ABB RAPID module: old_Module1.mod

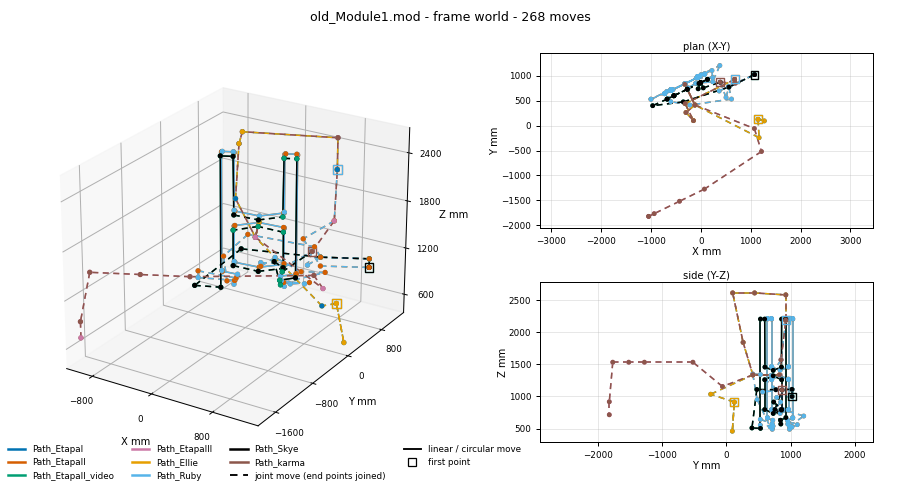
[picture p0: tool path of old_Module1.mod in frame world, 268 of 268 moves have a stored position in this frame; points joined in program order, loops and branches not executed]
MODULE Module1
	CONST robtarget Target_20_2:=[[0,0.000001,500],[0,0,1,-0.000000001],[-2,-1,0,0],[9E9,9E9,9E9,9E9,9E9,9E9]];
	CONST robtarget Target_10:=[[3.472963553,17.439983187,29.999999981],[0,0,1,-0.000000001],[-2,-1,0,0],[9E9,9E9,9E9,9E9,9E9,9E9]];
	CONST robtarget Target_20:=[[0,0.000001,500],[0,0,1,-0.000000001],[-2,-1,0,0],[9E9,9E9,9E9,9E9,9E9,9E9]];
	CONST robtarget Target_20_2_3:=[[355.257254851,-131.298701917,586.23338687],[0,0,1,-0.000000001],[-2,-1,0,0],[9E9,9E9,9E9,9E9,9E9,9E9]];
	CONST robtarget Target_30:=[[-728.668360128,-898.010521018,1225.921750474],[0.579227966,0.405579787,-0.5,-0.5],[0,0,0,0],[9E9,9E9,9E9,9E9,9E9,9E9]];
	CONST robtarget Target_30_3:=[[-1183.134430466,-884.095288461,1304.838955392],[0.579227966,0.405579787,-0.5,-0.5],[1,0,0,0],[9E9,9E9,9E9,9E9,9E9,9E9]];
	CONST robtarget Target_70:=[[-584.684106736,-1037.65235773,1745.210003217],[0.579227966,0.405579787,-0.5,-0.5],[0,0,0,4],[9E9,9E9,9E9,9E9,9E9,9E9]];
	CONST robtarget Target_80_2:=[[-242.789561942,-850.912741716,2444.405198949],[0.579227966,0.405579787,-0.5,-0.5],[1,0,0,4],[9E9,9E9,9E9,9E9,9E9,9E9]];
	CONST robtarget Target_80:=[[-616.524860071,-839.469393295,2509.303652393],[0.69636424,-0.122787804,0,-0.707106781],[0,-1,1,1],[9E9,9E9,9E9,9E9,9E9,9E9]];
	CONST robtarget Target_90:=[[-621.798393161,243.110506611,2288.046539347],[0.69636424,-0.122787804,0,-0.707106781],[0,-1,1,1],[9E9,9E9,9E9,9E9,9E9,9E9]];
	CONST robtarget Target_90_2:=[[-690.279328238,175.6699504,1905.572141463],[0.69636424,-0.122787804,0,-0.707106781],[0,-1,1,1],[9E9,9E9,9E9,9E9,9E9,9E9]];
	CONST robtarget Target_90_2_2:=[[690.970814762,851.051580359,1570.162539077],[0.225435439,0,0,-0.974258109],[0,0,1,1],[9E9,9E9,9E9,9E9,9E9,9E9]];
	CONST robtarget Target_90_2_2_3:=[[367.891360431,693.077349856,1324.929850073],[0,0.848311443,-0.529497588,0],[0,0,-1,0],[9E9,9E9,9E9,9E9,9E9,9E9]];
	CONST robtarget Target_90_2_2_3_2:=[[553.518951213,783.842563864,984.266783155],[0,0.848311443,-0.529497588,0],[0,0,-1,0],[9E9,9E9,9E9,9E9,9E9,9E9]];
	CONST robtarget Target_90_2_2_3_2_2:=[[1075.518835373,1022.097696077,1000],[0,0.848311443,-0.529497588,0],[0,0,-1,0],[9E9,9E9,9E9,9E9,9E9,9E9]];
	CONST robtarget Target_90_2_2_3_2_2_2:=[[1075.518835373,1022.097696077,1000],[0,0.848311443,-0.529497588,0],[0,0,-1,0],[9E9,9E9,9E9,9E9,9E9,9E9]];
	CONST robtarget Target_100:=[[1075.303889935,1021.965880074,1110.91287582],[0,0.848311443,-0.529497588,0],[0,0,-1,0],[9E9,9E9,9E9,9E9,9E9,9E9]];
	CONST robtarget Target_110:=[[561.343174474,770.657579762,1105.422922565],[0,0.848311443,-0.529497588,0],[0,0,-1,0],[9E9,9E9,9E9,9E9,9E9,9E9]];
	CONST robtarget Target_120:=[[614.35326876,531.541624289,1341.660223262],[0.630196274,-0.425266678,-0.564932078,-0.320706495],[0,0,1,0],[9E9,9E9,9E9,9E9,9E9,9E9]];
	CONST robtarget Target_130:=[[-220.756964436,411.144811502,1349.578986688],[0.630196274,-0.425266678,-0.564932078,-0.320706495],[1,1,0,1],[9E9,9E9,9E9,9E9,9E9,9E9]];
	CONST robtarget Target_140:=[[-603.640790819,480.038707024,951.826023694],[0.630196274,-0.425266678,-0.564932078,-0.320706495],[1,0,1,1],[9E9,9E9,9E9,9E9,9E9,9E9]];
	CONST robtarget Target_150:=[[-684.956865831,682.802213826,527.356838346],[0.630196274,-0.425266678,-0.564932078,-0.320706495],[1,0,1,1],[9E9,9E9,9E9,9E9,9E9,9E9]];
	CONST robtarget Target_160:=[[-600.231193595,724.230019574,538.596152517],[0.630196274,-0.425266678,-0.564932078,-0.320706495],[1,0,1,1],[9E9,9E9,9E9,9E9,9E9,9E9]];
	CONST robtarget Target_170:=[[-615.502782618,744.38841834,511.008322261],[0.630196274,-0.425266678,-0.564932078,-0.320706495],[1,0,1,1],[9E9,9E9,9E9,9E9,9E9,9E9]];
	CONST robtarget Target_180:=[[-605.289704553,715.096779867,490.071182954],[0.630196274,-0.425266678,-0.564932078,-0.320706495],[1,0,1,1],[9E9,9E9,9E9,9E9,9E9,9E9]];
	CONST robtarget Target_190:=[[-592.759513668,700.25774586,516.943595123],[0.630196274,-0.425266678,-0.564932078,-0.320706495],[1,0,1,1],[9E9,9E9,9E9,9E9,9E9,9E9]];
	CONST robtarget Target_200:=[[-600.231193595,724.230019574,538.596152517],[0.630196274,-0.425266678,-0.564932078,-0.320706495],[1,0,1,1],[9E9,9E9,9E9,9E9,9E9,9E9]];
	CONST robtarget Target_210:=[[-1000.069986007,528.723234139,554.74513186],[0.630196274,-0.425266678,-0.564932078,-0.320706495],[1,0,1,1],[9E9,9E9,9E9,9E9,9E9,9E9]];
	CONST robtarget Target_210_2:=[[-1000.069986007,528.723234139,644.473462045],[0.74632501,0.144907108,-0.626241041,0.172693565],[1,-1,2,1],[9E9,9E9,9E9,9E9,9E9,9E9]];
	CONST robtarget Target_220:=[[-574.244255672,714.673851005,578.901883612],[0.74632501,0.144907108,-0.626241041,0.172693565],[1,-2,-2,1],[9E9,9E9,9E9,9E9,9E9,9E9]];
	CONST robtarget Target_230:=[[-558.661492442,722.293261641,630.386873665],[0.74632501,0.144907108,-0.626241041,0.172693565],[1,-2,-2,1],[9E9,9E9,9E9,9E9,9E9,9E9]];
	CONST robtarget Target_240:=[[-721.925864829,642.46285692,662.431918782],[0.74632501,0.144907108,-0.626241041,0.172693565],[1,-1,-2,1],[9E9,9E9,9E9,9E9,9E9,9E9]];
	CONST robtarget Target_250:=[[-727.247702444,639.860669777,665.852120215],[0.74632501,0.144907108,-0.626241041,0.172693565],[1,-1,-2,1],[9E9,9E9,9E9,9E9,9E9,9E9]];
	CONST robtarget Target_260:=[[-729.349460263,638.832985813,672.279996312],[0.74632501,0.144907108,-0.626241041,0.172693565],[1,-1,-2,1],[9E9,9E9,9E9,9E9,9E9,9E9]];
	CONST robtarget Target_270:=[[-729.349460263,638.832985813,2203.889],[0.74632501,0.144907108,-0.626241041,0.172693565],[1,-1,-1,1],[9E9,9E9,9E9,9E9,9E9,9E9]];
	CONST robtarget Target_280:=[[-726.718231405,640.119562068,2210.960067812],[0.74632501,0.144907108,-0.626241041,0.172693565],[1,-1,-1,1],[9E9,9E9,9E9,9E9,9E9,9E9]];
	CONST robtarget Target_290:=[[-720.36588301,643.22563191,2213.889],[0.970550763,-0.019647992,0.084912189,0.22457759],[1,0,-2,1],[9E9,9E9,9E9,9E9,9E9,9E9]];
	CONST robtarget Target_300:=[[-603.579378711,700.33003116,2213.889],[0.970550763,-0.019647992,0.084912189,0.22457759],[1,0,-2,1],[9E9,9E9,9E9,9E9,9E9,9E9]];
	CONST robtarget Target_310:=[[-597.227030315,703.436101002,2210.960067812],[0.970550763,-0.019647992,0.084912189,0.22457759],[1,0,-2,1],[9E9,9E9,9E9,9E9,9E9,9E9]];
	CONST robtarget Target_320:=[[-594.595801457,704.722677256,2203.889],[0.970550763,-0.019647992,0.084912189,0.22457759],[1,0,-2,1],[9E9,9E9,9E9,9E9,9E9,9E9]];
	CONST robtarget Target_330:=[[-594.595801457,704.722677256,1467.279996312],[0.970550763,-0.019647992,0.084912189,0.22457759],[1,0,-2,1],[9E9,9E9,9E9,9E9,9E9,9E9]];
	CONST robtarget Target_340:=[[-592.494043638,705.75036122,1460.852120215],[0.970550763,-0.019647992,0.084912189,0.22457759],[1,0,-2,1],[9E9,9E9,9E9,9E9,9E9,9E9]];
	CONST robtarget Target_350:=[[-587.172206023,708.352548362,1457.431918782],[0.970550763,-0.019647992,0.084912189,0.22457759],[1,0,-2,1],[9E9,9E9,9E9,9E9,9E9,9E9]];
	CONST robtarget Target_360:=[[-323.528502026,837.264835131,1406.297094376],[0.970550763,-0.019647992,0.084912189,0.22457759],[1,0,-1,1],[9E9,9E9,9E9,9E9,9E9,9E9]];
	CONST robtarget Target_370:=[[-63.004761668,964.65157192,1457.431918782],[0.970550763,-0.019647992,0.084912189,0.22457759],[1,0,-1,1],[9E9,9E9,9E9,9E9,9E9,9E9]];
	CONST robtarget Target_380:=[[-57.682924053,967.253759063,1460.852120215],[0.970550763,-0.019647992,0.084912189,0.22457759],[1,0,-1,1],[9E9,9E9,9E9,9E9,9E9,9E9]];
	CONST robtarget Target_390:=[[-55.581166233,968.281443027,1467.279996312],[0.970550763,-0.019647992,0.084912189,0.22457759],[1,0,-1,1],[9E9,9E9,9E9,9E9,9E9,9E9]];
	CONST robtarget Target_400:=[[-55.581166233,968.281443027,2203.889],[0.970550763,-0.019647992,0.084912189,0.22457759],[1,0,-1,1],[9E9,9E9,9E9,9E9,9E9,9E9]];
	CONST robtarget Target_410:=[[-52.949937375,969.568019281,2210.960067812],[0.970550763,-0.019647992,0.084912189,0.22457759],[1,0,-1,1],[9E9,9E9,9E9,9E9,9E9,9E9]];
	CONST robtarget Target_420:=[[-46.59758898,972.674089123,2213.889],[0.970550763,-0.019647992,0.084912189,0.22457759],[1,0,-1,1],[9E9,9E9,9E9,9E9,9E9,9E9]];
	CONST robtarget Target_430:=[[70.188915319,1029.778488373,2213.889],[0.970550763,-0.019647992,0.084912189,0.22457759],[0,0,-1,1],[9E9,9E9,9E9,9E9,9E9,9E9]];
	CONST robtarget Target_440:=[[76.541263714,1032.884558215,2210.960067812],[0.970550763,-0.019647992,0.084912189,0.22457759],[0,0,-1,1],[9E9,9E9,9E9,9E9,9E9,9E9]];
	CONST robtarget Target_450:=[[79.172492573,1034.171134469,2203.889],[0.626241041,-0.172693565,0.74632501,0.144907108],[1,1,-2,1],[9E9,9E9,9E9,9E9,9E9,9E9]];
	CONST robtarget Target_460:=[[79.172492573,1034.171134469,672.279996312],[0.626241041,-0.172693565,0.74632501,0.144907108],[1,0,-1,1],[9E9,9E9,9E9,9E9,9E9,9E9]];
	CONST robtarget Target_470:=[[77.070734753,1033.143450506,665.852120215],[0.626241041,-0.172693565,0.74632501,0.144907108],[1,0,-1,1],[9E9,9E9,9E9,9E9,9E9,9E9]];
	CONST robtarget Target_480:=[[71.748897138,1030.541263363,662.431918782],[0.626241041,-0.172693565,0.74632501,0.144907108],[1,0,-1,1],[9E9,9E9,9E9,9E9,9E9,9E9]];
	CONST robtarget Target_490:=[[-91.515475248,950.710858642,630.386873665],[0.626241041,-0.172693565,0.74632501,0.144907108],[1,1,-1,1],[9E9,9E9,9E9,9E9,9E9,9E9]];
	CONST robtarget Target_500:=[[-82.17325952,955.27886605,571.409990938],[0.626241041,-0.172693565,0.74632501,0.144907108],[1,1,-1,1],[9E9,9E9,9E9,9E9,9E9,9E9]];
	CONST robtarget Target_500_2:=[[235.647161917,962.336296138,604.766182313],[0.626241041,-0.172693565,0.74632501,0.144907108],[0,0,-1,1],[9E9,9E9,9E9,9E9,9E9,9E9]];
	CONST robtarget Target_500_2_2:=[[222.398190082,1104.203348059,561.899220237],[0.320706496,-0.564932078,0.425266677,0.630196274],[0,1,-2,0],[9E9,9E9,9E9,9E9,9E9,9E9]];
	CONST robtarget Target_510:=[[4.592265391,1019.966932715,523.466438018],[0.425266678,-0.630196274,0.320706495,0.564932078],[0,1,-2,0],[9E9,9E9,9E9,9E9,9E9,9E9]];
	CONST robtarget Target_520:=[[-67.51635848,984.708409724,538.596152517],[0.425266678,-0.630196274,0.320706495,0.564932078],[0,1,-2,0],[9E9,9E9,9E9,9E9,9E9,9E9]];
	CONST robtarget Target_530:=[[-74.04786326,1009.140395264,511.008322261],[0.425266678,-0.630196274,0.320706495,0.564932078],[0,1,-2,0],[9E9,9E9,9E9,9E9,9E9,9E9]];
	CONST robtarget Target_540:=[[-57.20170243,983.09209564,490.071182954],[0.425266678,-0.630196274,0.320706495,0.564932078],[0,1,-2,0],[9E9,9E9,9E9,9E9,9E9,9E9]];
	CONST robtarget Target_550:=[[-53.184944606,964.090299134,516.943595123],[0.425266678,-0.630196274,0.320706495,0.564932078],[0,1,-2,0],[9E9,9E9,9E9,9E9,9E9,9E9]];
	CONST robtarget Target_560:=[[-67.51635848,984.708409724,538.596152517],[0.425266678,-0.630196274,0.320706495,0.564932078],[0,1,-2,0],[9E9,9E9,9E9,9E9,9E9,9E9]];
	CONST robtarget Target_570:=[[380.563228786,1203.803208398,695.774665043],[0.425266678,-0.630196274,0.320706495,0.564932078],[0,1,-2,0],[9E9,9E9,9E9,9E9,9E9,9E9]];
	CONST robtarget Target_580_3:=[[236.855316057,878.977367128,797.279996312],[0.626241041,-0.172693565,0.74632501,0.144907108],[0,0,-1,1],[9E9,9E9,9E9,9E9,9E9,9E9]];
	CONST robtarget Target_740:=[[-106.574951523,844.917671275,913.754533399],[0.626241041,-0.172693565,0.74632501,0.144907108],[1,1,-1,1],[9E9,9E9,9E9,9E9,9E9,9E9]];
	CONST robtarget Target_580_3_2:=[[-251.957733199,755.881530829,797.279996312],[0.626241041,-0.172693565,0.74632501,0.144907108],[1,1,-1,1],[9E9,9E9,9E9,9E9,9E9,9E9]];
	CONST robtarget Target_580:=[[-306.602704629,845.540941159,797.279996312],[0.626241041,-0.172693565,0.74632501,0.144907108],[1,1,-1,1],[9E9,9E9,9E9,9E9,9E9,9E9]];
	CONST robtarget Target_590:=[[-55.581166233,968.281443027,797.279996312],[0.626241041,-0.172693565,0.74632501,0.144907108],[1,1,-1,1],[9E9,9E9,9E9,9E9,9E9,9E9]];
	CONST robtarget Target_600:=[[-55.581166233,968.281443027,1260.498003688],[0.626241041,-0.172693565,0.74632501,0.144907108],[1,1,-1,1],[9E9,9E9,9E9,9E9,9E9,9E9]];
	CONST robtarget Target_610:=[[-57.682924053,967.253759063,1266.925879785],[0.626241041,-0.172693565,0.74632501,0.144907108],[1,1,-1,1],[9E9,9E9,9E9,9E9,9E9,9E9]];
	CONST robtarget Target_620:=[[-63.004761668,964.65157192,1270.346081218],[0.626241041,-0.172693565,0.74632501,0.144907108],[1,1,-1,1],[9E9,9E9,9E9,9E9,9E9,9E9]];
	CONST robtarget Target_630:=[[-326.648465665,835.739285151,1321.480905624],[0.626241041,-0.172693565,0.74632501,0.144907108],[1,1,-1,1],[9E9,9E9,9E9,9E9,9E9,9E9]];
	CONST robtarget Target_640:=[[-587.172206023,708.352548362,1270.346081218],[0.626241041,-0.172693565,0.74632501,0.144907108],[1,1,-1,1],[9E9,9E9,9E9,9E9,9E9,9E9]];
	CONST robtarget Target_650:=[[-592.494043638,705.75036122,1266.925879785],[0.626241041,-0.172693565,0.74632501,0.144907108],[1,1,-1,1],[9E9,9E9,9E9,9E9,9E9,9E9]];
	CONST robtarget Target_660:=[[-594.595801457,704.722677256,1260.498003688],[0.626241041,-0.172693565,0.74632501,0.144907108],[1,1,-1,1],[9E9,9E9,9E9,9E9,9E9,9E9]];
	CONST robtarget Target_670:=[[-594.595801457,704.722677256,797.279996312],[0.626241041,-0.172693565,0.74632501,0.144907108],[1,1,-1,1],[9E9,9E9,9E9,9E9,9E9,9E9]];
	CONST robtarget Target_680:=[[-592.494043638,705.75036122,790.852120215],[0.626241041,-0.172693565,0.74632501,0.144907108],[1,1,-1,1],[9E9,9E9,9E9,9E9,9E9,9E9]];
	CONST robtarget Target_690:=[[-587.172206023,708.352548362,787.431918782],[0.626241041,-0.172693565,0.74632501,0.144907108],[1,1,-1,1],[9E9,9E9,9E9,9E9,9E9,9E9]];
	CONST robtarget Target_700:=[[-323.528502026,837.264835131,736.297094376],[0.626241041,-0.172693565,0.74632501,0.144907108],[1,1,-1,1],[9E9,9E9,9E9,9E9,9E9,9E9]];
	CONST robtarget Target_710:=[[-63.004761668,964.65157192,787.431918782],[0.626241041,-0.172693565,0.74632501,0.144907108],[1,1,-1,1],[9E9,9E9,9E9,9E9,9E9,9E9]];
	CONST robtarget Target_720:=[[-57.682924053,967.253759063,790.852120215],[0.626241041,-0.172693565,0.74632501,0.144907108],[1,1,-1,1],[9E9,9E9,9E9,9E9,9E9,9E9]];
	CONST robtarget Target_730:=[[-55.581166233,968.281443027,797.279996312],[0.626241041,-0.172693565,0.74632501,0.144907108],[1,1,-1,1],[9E9,9E9,9E9,9E9,9E9,9E9]];
	CONST robtarget Target_730_2:=[[-4.129380996,863.055327059,797.279996312],[0.626241041,-0.172693565,0.74632501,0.144907108],[1,1,-1,1],[9E9,9E9,9E9,9E9,9E9,9E9]];
	CONST robtarget Target_130_2:=[[389.997020927,869.040623857,1101.572770211],[0.630196274,-0.425266678,-0.564932078,-0.320706495],[0,1,0,0],[9E9,9E9,9E9,9E9,9E9,9E9]];
	CONST robtarget Target_120_2:=[[504.928038476,563.849286682,1069.091100494],[0,0.848311443,-0.529497588,0],[0,0,-1,0],[9E9,9E9,9E9,9E9,9E9,9E9]];
	CONST robtarget Target_110_2:=[[561.343174474,770.657579762,1105.422922565],[0,0.848311443,-0.529497588,0],[0,0,-1,0],[9E9,9E9,9E9,9E9,9E9,9E9]];
	CONST robtarget Target_90_2_2_3_2_2_2_2:=[[1075.518835373,1022.097696077,1000],[0,0.848311443,-0.529497588,0],[0,0,-1,0],[9E9,9E9,9E9,9E9,9E9,9E9]];
	CONST robtarget Target_100_2:=[[1075.303889935,1021.965880074,1110.91287582],[0,0.848311443,-0.529497588,0],[0,0,-1,0],[9E9,9E9,9E9,9E9,9E9,9E9]];
	CONST robtarget Target_110_3:=[[561.343174474,770.657579762,1105.422922565],[0,0.848311443,-0.529497588,0],[0,0,-1,0],[9E9,9E9,9E9,9E9,9E9,9E9]];
	CONST robtarget Target_120_3:=[[-352.181570531,474.725664361,1108.429867517],[0.630196274,-0.425266678,-0.564932078,-0.320706495],[1,-2,-1,0],[9E9,9E9,9E9,9E9,9E9,9E9]];
	CONST robtarget Target_130_3:=[[-965.595492909,398.655755176,510.210088752],[0.630196274,-0.425266678,-0.564932078,-0.320706495],[1,-2,-1,0],[9E9,9E9,9E9,9E9,9E9,9E9]];
	CONST robtarget Target_260_2:=[[-676.765426106,531.291262028,504.173173014],[0.630196274,-0.425266678,-0.564932078,-0.320706495],[1,-2,-1,0],[9E9,9E9,9E9,9E9,9E9,9E9]];
	CONST robtarget Target_270_2:=[[-676.765426106,531.291262028,2203.889],[0.630196274,-0.425266678,-0.564932078,-0.320706495],[1,-1,-2,0],[9E9,9E9,9E9,9E9,9E9,9E9]];
	CONST robtarget Target_320_2:=[[-542.0117673,597.180953471,2203.889],[0.630196274,-0.425266678,-0.564932078,-0.320706495],[1,-1,-2,0],[9E9,9E9,9E9,9E9,9E9,9E9]];
	CONST robtarget Target_350_2:=[[-534.588171866,600.810824577,1457.431918782],[0.630196274,-0.425266678,-0.564932078,-0.320706495],[1,-1,-1,0],[9E9,9E9,9E9,9E9,9E9,9E9]];
	CONST robtarget Target_360_2:=[[-270.944467869,729.723111346,1406.297094376],[0.630196274,-0.425266678,-0.564932078,-0.320706495],[1,-1,-1,1],[9E9,9E9,9E9,9E9,9E9,9E9]];
	CONST robtarget Target_370_2:=[[-10.420727511,857.109848135,1457.431918782],[0.630196274,-0.425266678,-0.564932078,-0.320706495],[0,-1,-1,1],[9E9,9E9,9E9,9E9,9E9,9E9]];
	CONST robtarget Target_400_2:=[[-2.997132076,860.739719242,2203.889],[0.630196274,-0.425266678,-0.564932078,-0.320706495],[0,-2,-1,1],[9E9,9E9,9E9,9E9,9E9,9E9]];
	CONST robtarget Target_450_2:=[[131.75652673,926.629410684,2203.889],[0.630196274,-0.425266678,-0.564932078,-0.320706495],[0,-2,-1,1],[9E9,9E9,9E9,9E9,9E9,9E9]];
	CONST robtarget Target_460_2:=[[131.75652673,926.629410684,672.279996312],[0.630196274,-0.425266678,-0.564932078,-0.320706495],[0,-1,-2,1],[9E9,9E9,9E9,9E9,9E9,9E9]];
	CONST robtarget Target_490_2:=[[-38.931441091,843.169134857,630.386873665],[0.630196274,-0.425266678,-0.564932078,-0.320706495],[0,-1,-2,1],[9E9,9E9,9E9,9E9,9E9,9E9]];
	CONST robtarget Target_500_3:=[[-29.589225363,847.737142265,571.409990938],[0.630196274,-0.425266678,-0.564932078,-0.320706495],[0,-1,-2,1],[9E9,9E9,9E9,9E9,9E9,9E9]];
	CONST robtarget Target_740_2:=[[-53.990917366,737.37594749,913.754533399],[0.630196274,-0.425266678,-0.564932078,-0.320706495],[0,-1,-2,1],[9E9,9E9,9E9,9E9,9E9,9E9]];
	CONST robtarget Target_590_2:=[[-2.997132076,860.739719242,797.279996312],[0.630196274,-0.425266678,-0.564932078,-0.320706495],[0,-1,-2,1],[9E9,9E9,9E9,9E9,9E9,9E9]];
	CONST robtarget Target_600_2:=[[-2.997132076,860.739719242,1260.498003688],[0.630196274,-0.425266678,-0.564932078,-0.320706495],[0,-1,-2,1],[9E9,9E9,9E9,9E9,9E9,9E9]];
	CONST robtarget Target_630_2:=[[-274.064431508,728.197561366,1321.480905624],[0.630196274,-0.425266678,-0.564932078,-0.320706495],[1,-1,-2,1],[9E9,9E9,9E9,9E9,9E9,9E9]];
	CONST robtarget Target_660_2:=[[-542.0117673,597.180953471,1260.498003688],[0.630196274,-0.425266678,-0.564932078,-0.320706495],[1,-2,-1,0],[9E9,9E9,9E9,9E9,9E9,9E9]];
	CONST robtarget Target_670_2:=[[-542.0117673,597.180953471,797.279996312],[0.630196274,-0.425266678,-0.564932078,-0.320706495],[1,-2,-1,0],[9E9,9E9,9E9,9E9,9E9,9E9]];
	CONST robtarget Target_700_2:=[[-270.944467869,729.723111346,736.297094376],[0.630196274,-0.425266678,-0.564932078,-0.320706495],[1,-1,-2,1],[9E9,9E9,9E9,9E9,9E9,9E9]];
	CONST robtarget Target_710_2:=[[-10.420727511,857.109848135,787.431918782],[0.630196274,-0.425266678,-0.564932078,-0.320706495],[0,-1,-2,1],[9E9,9E9,9E9,9E9,9E9,9E9]];
	CONST robtarget Target_730_3:=[[-2.997132076,860.739719242,797.279996312],[0.630196274,-0.425266678,-0.564932078,-0.320706495],[0,-1,-2,1],[9E9,9E9,9E9,9E9,9E9,9E9]];
	CONST robtarget Target_730_2_2:=[[48.454653161,755.513603274,797.279996312],[0.630196274,-0.425266678,-0.564932078,-0.320706495],[0,-1,-2,1],[9E9,9E9,9E9,9E9,9E9,9E9]];
	CONST robtarget Target_130_2_2:=[[389.997020927,869.040623857,1101.572770211],[0.630196274,-0.425266678,-0.564932078,-0.320706495],[0,-1,-2,1],[9E9,9E9,9E9,9E9,9E9,9E9]];
	CONST robtarget Target_130_2_2_2:=[[389.997020927,869.040623857,1101.572770211],[0.630196274,-0.425266678,-0.564932078,-0.320706495],[0,-1,-2,1],[9E9,9E9,9E9,9E9,9E9,9E9]];
	CONST robtarget Target_90_2_2_2:=[[690.970814762,851.051580359,1570.162539077],[0.225435439,0,0,-0.974258109],[0,0,1,1],[9E9,9E9,9E9,9E9,9E9,9E9]];
	CONST robtarget Target_90_2_3:=[[677.216886302,925.105208889,2185.609751442],[0.225435439,0,0,-0.974258109],[0,0,1,1],[9E9,9E9,9E9,9E9,9E9,9E9]];
	CONST robtarget Target_90_2_4:=[[677.216886302,925.105208889,2185.609751442],[0.225435439,0,0,-0.974258109],[0,0,1,1],[9E9,9E9,9E9,9E9,9E9,9E9]];
	CONST robtarget Target_90_3:=[[677.216886303,925.105208888,2579.975738982],[0.225435439,0,0,-0.974258109],[0,0,1,1],[9E9,9E9,9E9,9E9,9E9,9E9]];
	CONST robtarget Target_80_3:=[[-315.067708607,439.913739054,2610.344805668],[0.225435439,0,0,-0.974258109],[1,0,0,1],[9E9,9E9,9E9,9E9,9E9,9E9]];
	CONST robtarget Target_80_2_2:=[[-148.366452112,98.986292765,2610.344805667],[0.159406928,0.159406928,-0.688904515,-0.688904516],[1,0,0,4],[9E9,9E9,9E9,9E9,9E9,9E9]];
	CONST robtarget Target_70_2:=[[-297.408117168,261.539979913,1840.929204997],[0.159406928,0.159406928,-0.688904515,-0.688904516],[0,0,0,4],[9E9,9E9,9E9,9E9,9E9,9E9]];
	CONST robtarget Target_30_2:=[[-117.985307131,412.947477324,1336.176966578],[0.159406928,0.159406928,-0.688904515,-0.688904516],[0,0,0,0],[9E9,9E9,9E9,9E9,9E9,9E9]];
	CONST robtarget Target_30_3_2:=[[-320.695795916,827.518853271,1336.176966578],[0.159406928,0.159406928,-0.688904515,-0.688904516],[1,0,0,0],[9E9,9E9,9E9,9E9,9E9,9E9]];
	CONST robtarget Target_30_2_2:=[[-117.985307131,412.947477324,1336.176966578],[0.159406928,0.159406928,-0.688904515,-0.688904516],[0,0,0,0],[9E9,9E9,9E9,9E9,9E9,9E9]];
	CONST robtarget Target_30_2_3:=[[1072.781898944,-59.825918958,1155.239486671],[0.374411334,0.374411335,0.599846774,0.599846775],[-1,1,-1,0],[9E9,9E9,9E9,9E9,9E9,9E9]];
	CONST robtarget Target_30_2_3_2:=[[1215.425844801,-519.48484737,1533.087792477],[0.374411334,0.374411335,0.599846774,0.599846775],[-1,1,-1,0],[9E9,9E9,9E9,9E9,9E9,9E9]];
	CONST robtarget Target_30_2_3_2_2:=[[71.368530681,-1273.53877769,1533.087792477],[0.688904515,0.688904516,0.159406928,0.159406928],[-2,1,-1,0],[9E9,9E9,9E9,9E9,9E9,9E9]];
	CONST robtarget Target_30_2_3_2_2_2:=[[-427.431513587,-1517.434055188,1533.087792477],[0.000000001,0.974258109,0.225435439,0],[-2,-1,0,0],[9E9,9E9,9E9,9E9,9E9,9E9]];
	CONST robtarget Target_30_2_3_2_2_2_2:=[[-935.838539063,-1766.02680089,1533.087792477],[-0.000000001,0.974258109,0.225435439,0],[-2,0,0,0],[9E9,9E9,9E9,9E9,9E9,9E9]];
	CONST robtarget Target_30_2_3_2_2_2_2_2:=[[-1046.370183316,-1820.072798594,917.887564527],[-0.000000001,0.974258109,0.225435439,0],[-2,0,0,0],[9E9,9E9,9E9,9E9,9E9,9E9]];
	CONST robtarget Target_30_2_3_2_2_2_2_2_2:=[[-1046.370183316,-1820.072798594,715.608584776],[-0.000000001,0.974258109,0.225435439,0],[-2,0,0,0],[9E9,9E9,9E9,9E9,9E9,9E9]];
	PROC Path_EtapaI()
	    MoveJ Target_20_2,v500,z100,Tooldata_TCP_VAC\WObj:=Workobject_EtapaI;
	    MoveJ Target_10,v400,z100,Tooldata_TCP_VAC\WObj:=Workobject_EtapaI;
	    MoveJ Target_20,v500,z100,Tooldata_TCP_VAC\WObj:=Workobject_EtapaI;
	    MoveJ Target_20_2_3,v500,z100,Tooldata_TCP_VAC\WObj:=Workobject_EtapaI;
	    MoveJ Target_30,v500,z100,Tooldata_TCP_VAC\WObj:=Workobject_EtapaI;
	    MoveJ Target_30_3,v500,z100,Tooldata_TCP_VAC\WObj:=Workobject_EtapaI;
	    MoveJ Target_30,v500,z100,Tooldata_TCP_VAC\WObj:=Workobject_EtapaI;
	    MoveJ Target_70,v500,z100,Tooldata_TCP_VAC\WObj:=Workobject_EtapaI;
	    MoveJ Target_80_2,v500,z100,Tooldata_TCP_VAC\WObj:=Workobject_EtapaI;
	    MoveJ Target_80,v500,z100,Tooldata_TCP_VAC\WObj:=Workobject_EtapaI;
	    MoveJ Target_90,v500,z100,Tooldata_TCP_VAC\WObj:=Workobject_EtapaI;
	    MoveJ Target_90_2,v500,z100,Tooldata_TCP_VAC\WObj:=Workobject_EtapaI;
	ENDPROC
	PROC Path_EtapaII()
	    MoveJ Target_90_2,v500,z100,Tooldata_TCP_VAC\WObj:=Workobject_EtapaI;
	    MoveJ Target_90_2_2,v500,z100,Flansa_Cuplare\WObj:=Workobject_EtapaII;
	    MoveJ Target_90_2_2_3,v500,z100,Flansa_Cuplare\WObj:=Workobject_EtapaII;
	    MoveJ Target_90_2_2_3_2,v500,z100,Flansa_Cuplare\WObj:=Workobject_EtapaII;
	    MoveJ Target_90_2_2_3_2_2,v500,z100,Flansa_Cuplare\WObj:=Workobject_EtapaII;
	    MoveJ Target_90_2_2_3_2_2_2,v500,z100,Flansa_Cuplare\WObj:=Workobject_EtapaII;
	    MoveJ Target_100,v500,z100,Flansa_Cuplare\WObj:=Workobject_EtapaII;
	    MoveJ Target_110,v500,z100,Flansa_Cuplare\WObj:=Workobject_EtapaII;
	    MoveJ Target_120,v500,z100,Flansa_Cuplare\WObj:=Workobject_EtapaII;
	    MoveJ Target_130,v500,z100,Flansa_Cuplare\WObj:=Workobject_EtapaII;
	    MoveJ Target_140,v500,z100,Flansa_Cuplare\WObj:=Workobject_EtapaII;
	    MoveJ Target_150,v1000,z100,Tooldata_TCP_ATI\WObj:=Workobject_EtapaII;
	    MoveJ Target_160,v1000,z100,Tooldata_TCP_ATI\WObj:=Workobject_EtapaII;
	    MoveC Target_170,Target_180,v1000,z100,Tooldata_TCP_ATI\WObj:=Workobject_EtapaII;
	    MoveC Target_190,Target_200,v1000,z100,Tooldata_TCP_ATI\WObj:=Workobject_EtapaII;
	    MoveJ Target_210,v1000,z100,Tooldata_TCP_ATI\WObj:=Workobject_EtapaII;
	    MoveJ Target_210_2,v1000,z100,Tooldata_TCP_ATI\WObj:=Workobject_EtapaII;
	    MoveJ Target_220,v1000,z100,Tooldata_TCP_ATI\WObj:=Workobject_EtapaII;
	    MoveL Target_230,v1000,z100,Tooldata_TCP_ATI\WObj:=Workobject_EtapaII;
	    MoveL Target_240,v1000,z100,Tooldata_TCP_ATI\WObj:=Workobject_EtapaII;
	    MoveL Target_250,v1000,z100,Tooldata_TCP_ATI\WObj:=Workobject_EtapaII;
	    MoveL Target_260,v1000,z100,Tooldata_TCP_ATI\WObj:=Workobject_EtapaII;
	    MoveL Target_270,v1000,z100,Tooldata_TCP_ATI\WObj:=Workobject_EtapaII;
	    MoveL Target_280,v1000,z100,Tooldata_TCP_ATI\WObj:=Workobject_EtapaII;
	    MoveL Target_290,v1000,z100,Tooldata_TCP_ATI\WObj:=Workobject_EtapaII;
	    MoveL Target_300,v1000,z100,Tooldata_TCP_ATI\WObj:=Workobject_EtapaII;
	    MoveL Target_310,v1000,z100,Tooldata_TCP_ATI\WObj:=Workobject_EtapaII;
	    MoveL Target_320,v1000,z100,Tooldata_TCP_ATI\WObj:=Workobject_EtapaII;
	    MoveL Target_330,v1000,z100,Tooldata_TCP_ATI\WObj:=Workobject_EtapaII;
	    MoveL Target_340,v1000,z100,Tooldata_TCP_ATI\WObj:=Workobject_EtapaII;
	    MoveL Target_350,v1000,z100,Tooldata_TCP_ATI\WObj:=Workobject_EtapaII;
	    MoveL Target_360,v1000,z100,Tooldata_TCP_ATI\WObj:=Workobject_EtapaII;
	    MoveL Target_370,v1000,z100,Tooldata_TCP_ATI\WObj:=Workobject_EtapaII;
	    MoveL Target_380,v1000,z100,Tooldata_TCP_ATI\WObj:=Workobject_EtapaII;
	    MoveL Target_390,v1000,z100,Tooldata_TCP_ATI\WObj:=Workobject_EtapaII;
	    MoveL Target_400,v1000,z100,Tooldata_TCP_ATI\WObj:=Workobject_EtapaII;
	    MoveL Target_410,v1000,z100,Tooldata_TCP_ATI\WObj:=Workobject_EtapaII;
	    MoveL Target_420,v1000,z100,Tooldata_TCP_ATI\WObj:=Workobject_EtapaII;
	    MoveL Target_430,v1000,z100,Tooldata_TCP_ATI\WObj:=Workobject_EtapaII;
	    MoveJ Target_440,v1000,z100,Tooldata_TCP_ATI\WObj:=Workobject_EtapaII;
	    MoveJ Target_450,v1000,z100,Tooldata_TCP_ATI\WObj:=Workobject_EtapaII;
	    MoveL Target_460,v1000,z100,Tooldata_TCP_ATI\WObj:=Workobject_EtapaII;
	    MoveL Target_470,v1000,z100,Tooldata_TCP_ATI\WObj:=Workobject_EtapaII;
	    MoveL Target_480,v1000,z100,Tooldata_TCP_ATI\WObj:=Workobject_EtapaII;
	    MoveL Target_490,v1000,z100,Tooldata_TCP_ATI\WObj:=Workobject_EtapaII;
	    MoveL Target_500,v1000,z100,Tooldata_TCP_ATI\WObj:=Workobject_EtapaII;
	    MoveJ Target_500_2,v1000,z100,Tooldata_TCP_ATI\WObj:=Workobject_EtapaII;
	    MoveJ Target_500_2_2,v1000,z100,Tooldata_TCP_ATI\WObj:=Workobject_EtapaII;
	    MoveJ Target_510,v1000,z100,Tooldata_TCP_ATI\WObj:=Workobject_EtapaII;
	    MoveJ Target_520,v1000,z100,Tooldata_TCP_ATI\WObj:=Workobject_EtapaII;
	    MoveC Target_530,Target_540,v1000,z100,Tooldata_TCP_ATI\WObj:=Workobject_EtapaII;
	    MoveC Target_550,Target_560,v1000,z100,Tooldata_TCP_ATI\WObj:=Workobject_EtapaII;
	    MoveJ Target_570,v1000,z100,Tooldata_TCP_ATI\WObj:=Workobject_EtapaII;
	    MoveJ Target_580_3,v1000,z100,Tooldata_TCP_ATI\WObj:=Workobject_EtapaII;
	    MoveJ Target_740,v1000,z100,Tooldata_TCP_ATI\WObj:=Workobject_EtapaII;
	    MoveJ Target_580_3_2,v1000,z100,Tooldata_TCP_ATI\WObj:=Workobject_EtapaII;
	    MoveJ Target_580,v1000,z100,Tooldata_TCP_ATI\WObj:=Workobject_EtapaII;
	    MoveJ Target_590,v1000,z100,Tooldata_TCP_ATI\WObj:=Workobject_EtapaII;
	    MoveL Target_600,v1000,z100,Tooldata_TCP_ATI\WObj:=Workobject_EtapaII;
	    MoveL Target_610,v1000,z100,Tooldata_TCP_ATI\WObj:=Workobject_EtapaII;
	    MoveL Target_620,v1000,z100,Tooldata_TCP_ATI\WObj:=Workobject_EtapaII;
	    MoveL Target_630,v1000,z100,Tooldata_TCP_ATI\WObj:=Workobject_EtapaII;
	    MoveL Target_640,v1000,z100,Tooldata_TCP_ATI\WObj:=Workobject_EtapaII;
	    MoveL Target_650,v1000,z100,Tooldata_TCP_ATI\WObj:=Workobject_EtapaII;
	    MoveL Target_660,v1000,z100,Tooldata_TCP_ATI\WObj:=Workobject_EtapaII;
	    MoveL Target_670,v1000,z100,Tooldata_TCP_ATI\WObj:=Workobject_EtapaII;
	    MoveL Target_680,v1000,z100,Tooldata_TCP_ATI\WObj:=Workobject_EtapaII;
	    MoveL Target_690,v1000,z100,Tooldata_TCP_ATI\WObj:=Workobject_EtapaII;
	    MoveL Target_700,v1000,z100,Tooldata_TCP_ATI\WObj:=Workobject_EtapaII;
	    MoveL Target_710,v1000,z100,Tooldata_TCP_ATI\WObj:=Workobject_EtapaII;
	    MoveL Target_720,v1000,z100,Tooldata_TCP_ATI\WObj:=Workobject_EtapaII;
	    MoveL Target_730,v1000,z100,Tooldata_TCP_ATI\WObj:=Workobject_EtapaII;
	    MoveJ Target_730_2,v1000,z100,Tooldata_TCP_ATI\WObj:=Workobject_EtapaII;
	    MoveJ Target_130_2,v500,z100,Flansa_Cuplare\WObj:=Workobject_EtapaII;
	    MoveJ Target_120_2,v500,z100,Flansa_Cuplare\WObj:=Workobject_EtapaII;
	    MoveJ Target_110_2,v500,z100,Flansa_Cuplare\WObj:=Workobject_EtapaII;
	    MoveJ Target_100,v500,z100,Flansa_Cuplare\WObj:=Workobject_EtapaII;
	ENDPROC
	PROC Path_EtapaII_video()
	    MoveJ Target_90_2_2_3_2_2_2_2,v500,z100,Flansa_Cuplare\WObj:=Workobject_EtapaII_video;
	    MoveJ Target_100_2,v500,z100,Flansa_Cuplare\WObj:=Workobject_EtapaII_video;
	    MoveJ Target_110_3,v500,z100,Flansa_Cuplare\WObj:=Workobject_EtapaII_video;
	    MoveJ Target_120_3,v500,z100,Flansa_Cuplare\WObj:=Workobject_EtapaII_video;
	    MoveJ Target_130_3,v500,z50,Flansa_Cuplare\WObj:=Workobject_EtapaII_video;
	    MoveJ Target_260_2,v100,z50,Flansa_Cuplare\WObj:=Workobject_EtapaII_video;
	    MoveL Target_270_2,v200,z50,Flansa_Cuplare\WObj:=Workobject_EtapaII_video;
	    MoveL Target_320_2,v1000,z100,Flansa_Cuplare\WObj:=Workobject_EtapaII_video;
	    MoveL Target_350_2,v300,z30,Flansa_Cuplare\WObj:=Workobject_EtapaII_video;
	    MoveJ Target_360_2,v300,z30,Flansa_Cuplare\WObj:=Workobject_EtapaII_video;
	    MoveJ Target_370_2,v300,z30,Flansa_Cuplare\WObj:=Workobject_EtapaII_video;
	    MoveL Target_400_2,v300,z30,Flansa_Cuplare\WObj:=Workobject_EtapaII_video;
	    MoveJ Target_450_2,v300,z30,Flansa_Cuplare\WObj:=Workobject_EtapaII_video;
	    MoveL Target_460_2,v300,z30,Flansa_Cuplare\WObj:=Workobject_EtapaII_video;
	    MoveL Target_490_2,v300,z30,Flansa_Cuplare\WObj:=Workobject_EtapaII_video;
	    MoveL Target_500_3,v300,z30,Flansa_Cuplare\WObj:=Workobject_EtapaII_video;
	    MoveJ Target_740_2,v400,z20,Flansa_Cuplare\WObj:=Workobject_EtapaII_video;
	    MoveJ Target_590_2,v300,z30,Flansa_Cuplare\WObj:=Workobject_EtapaII_video;
	    MoveL Target_600_2,v300,z30,Flansa_Cuplare\WObj:=Workobject_EtapaII_video;
	    MoveJ Target_630_2,v300,z30,Flansa_Cuplare\WObj:=Workobject_EtapaII_video;
	    MoveJ Target_660_2,v300,z30,Flansa_Cuplare\WObj:=Workobject_EtapaII_video;
	    MoveL Target_670_2,v300,z30,Flansa_Cuplare\WObj:=Workobject_EtapaII_video;
	    MoveJ Target_700_2,v300,z30,Flansa_Cuplare\WObj:=Workobject_EtapaII_video;
	    MoveJ Target_710_2,v300,z30,Flansa_Cuplare\WObj:=Workobject_EtapaII_video;
	    MoveL Target_730_3,v300,z30,Flansa_Cuplare\WObj:=Workobject_EtapaII_video;
	    MoveJ Target_730_2_2,v300,z30,Flansa_Cuplare\WObj:=Workobject_EtapaII_video;
	    MoveJ Target_130_2_2,v300,z30,Flansa_Cuplare\WObj:=Workobject_EtapaII_video;
	ENDPROC
	PROC Path_EtapaIII()
	    MoveJ Target_130_2_2_2,v400,z30,Flansa_Cuplare\WObj:=Workobject_EtapaIII;
	    MoveJ Target_90_2_2_2,v400,z30,Flansa_Cuplare\WObj:=Workobject_EtapaIII;
	    MoveJ Target_90_2_3,v400,z30,Tooldata_TCP_VAC\WObj:=Workobject_EtapaIII;
	    MoveJ Target_90_2_4,v400,z30,Tooldata_TCP_VAC\WObj:=Workobject_EtapaIII;
	    MoveJ Target_90_3,v400,z30,Tooldata_TCP_VAC\WObj:=Workobject_EtapaIII;
	    MoveJ Target_80_3,v400,z30,Tooldata_TCP_VAC\WObj:=Workobject_EtapaIII;
	    MoveJ Target_80_2_2,v400,z30,Tooldata_TCP_VAC\WObj:=Workobject_EtapaIII;
	    MoveJ Target_70_2,v400,z30,Tooldata_TCP_VAC\WObj:=Workobject_EtapaIII;
	    MoveJ Target_30_2,v150,z10,Tooldata_TCP_VAC\WObj:=Workobject_EtapaIII;
	    MoveL Target_30_3_2,v150,z10,Tooldata_TCP_VAC\WObj:=Workobject_EtapaIII;
	    MoveL Target_30_2_2,v150,z10,Tooldata_TCP_VAC\WObj:=Workobject_EtapaIII;
	    MoveJ Target_30_2_3,v300,z30,Tooldata_TCP_VAC\WObj:=Workobject_EtapaIII;
	    MoveJ Target_30_2_3_2,v300,z30,Tooldata_TCP_VAC\WObj:=Workobject_EtapaIII;
	    MoveJ Target_30_2_3_2_2,v300,z30,Tooldata_TCP_VAC\WObj:=Workobject_EtapaIII;
	    MoveJ Target_30_2_3_2_2_2,v300,z30,Tooldata_TCP_VAC\WObj:=Workobject_EtapaIII;
	    MoveJ Target_30_2_3_2_2_2_2,v300,z30,Tooldata_TCP_VAC\WObj:=Workobject_EtapaIII;
	    MoveJ Target_30_2_3_2_2_2_2_2,v300,z30,Tooldata_TCP_VAC\WObj:=Workobject_EtapaIII;
	    MoveJ Target_30_2_3_2_2_2_2_2_2,v300,z30,Tooldata_TCP_VAC\WObj:=Workobject_EtapaIII;
	ENDPROC
	PROC Path_10()

	ENDPROC
	PROC Path_Ellie()
	    MoveJ Target_20_2,v500,z100,Tooldata_TCP_VAC\WObj:=Workobject_ellie;
	    MoveJ Target_10,v400,z100,Tooldata_TCP_VAC\WObj:=Workobject_ellie;
	    MoveJ Target_20,v500,z100,Tooldata_TCP_VAC\WObj:=Workobject_ellie;
	    MoveJ Target_20_2_3,v500,z100,Tooldata_TCP_VAC\WObj:=Workobject_ellie;
	    MoveJ Target_30,v500,z100,Tooldata_TCP_VAC\WObj:=Workobject_ellie;
	    MoveJ Target_30_3,v500,z100,Tooldata_TCP_VAC\WObj:=Workobject_ellie;
	    MoveJ Target_30,v500,z100,Tooldata_TCP_VAC\WObj:=Workobject_ellie;
	    MoveJ Target_70,v500,z100,Tooldata_TCP_VAC\WObj:=Workobject_ellie;
	    MoveJ Target_80_2,v500,z100,Tooldata_TCP_VAC\WObj:=Workobject_ellie;
	    MoveJ Target_80,v500,z100,Tooldata_TCP_VAC\WObj:=Workobject_ellie;
	    MoveJ Target_90,v500,z100,Tooldata_TCP_VAC\WObj:=Workobject_ellie;
	    MoveJ Target_90_2,v500,z100,Tooldata_TCP_VAC\WObj:=Workobject_ellie;
	ENDPROC
	PROC Path_Ruby()
	    MoveJ Target_90_2,v500,z100,Tooldata_TCP_VAC\WObj:=Workobject_ellie;
	    MoveJ Target_90_2_2,v500,z100,Flansa_Cuplare\WObj:=Workobject_ruby;
	    MoveJ Target_90_2_2_3,v500,z100,Flansa_Cuplare\WObj:=Workobject_ruby;
	    MoveJ Target_90_2_2_3_2,v500,z100,Flansa_Cuplare\WObj:=Workobject_ruby;
	    MoveJ Target_90_2_2_3_2_2,v500,z100,Flansa_Cuplare\WObj:=Workobject_ruby;
	    MoveJ Target_90_2_2_3_2_2_2,v500,z100,Flansa_Cuplare\WObj:=Workobject_ruby;
	    MoveJ Target_100,v500,z100,Flansa_Cuplare\WObj:=Workobject_ruby;
	    MoveJ Target_110,v500,z100,Flansa_Cuplare\WObj:=Workobject_ruby;
	    MoveJ Target_120,v500,z100,Flansa_Cuplare\WObj:=Workobject_ruby;
	    MoveJ Target_130,v500,z100,Flansa_Cuplare\WObj:=Workobject_ruby;
	    MoveJ Target_140,v500,z100,Flansa_Cuplare\WObj:=Workobject_ruby;
	    MoveJ Target_150,v1000,z100,Tooldata_TCP_ATI\WObj:=Workobject_ruby;
	    MoveJ Target_160,v1000,z100,Tooldata_TCP_ATI\WObj:=Workobject_ruby;
	    MoveC Target_170,Target_180,v1000,z100,Tooldata_TCP_ATI\WObj:=Workobject_ruby;
	    MoveC Target_190,Target_200,v1000,z100,Tooldata_TCP_ATI\WObj:=Workobject_ruby;
	    MoveJ Target_210,v1000,z100,Tooldata_TCP_ATI\WObj:=Workobject_ruby;
	    MoveJ Target_210_2,v1000,z100,Tooldata_TCP_ATI\WObj:=Workobject_ruby;
	    MoveJ Target_220,v1000,z100,Tooldata_TCP_ATI\WObj:=Workobject_ruby;
	    MoveL Target_230,v1000,z100,Tooldata_TCP_ATI\WObj:=Workobject_ruby;
	    MoveL Target_240,v1000,z100,Tooldata_TCP_ATI\WObj:=Workobject_ruby;
	    MoveL Target_250,v1000,z100,Tooldata_TCP_ATI\WObj:=Workobject_ruby;
	    MoveL Target_260,v1000,z100,Tooldata_TCP_ATI\WObj:=Workobject_ruby;
	    MoveL Target_270,v1000,z100,Tooldata_TCP_ATI\WObj:=Workobject_ruby;
	    MoveL Target_280,v1000,z100,Tooldata_TCP_ATI\WObj:=Workobject_ruby;
	    MoveL Target_290,v1000,z100,Tooldata_TCP_ATI\WObj:=Workobject_ruby;
	    MoveL Target_300,v1000,z100,Tooldata_TCP_ATI\WObj:=Workobject_ruby;
	    MoveL Target_310,v1000,z100,Tooldata_TCP_ATI\WObj:=Workobject_ruby;
	    MoveL Target_320,v1000,z100,Tooldata_TCP_ATI\WObj:=Workobject_ruby;
	    MoveL Target_330,v1000,z100,Tooldata_TCP_ATI\WObj:=Workobject_ruby;
	    MoveL Target_340,v1000,z100,Tooldata_TCP_ATI\WObj:=Workobject_ruby;
	    MoveL Target_350,v1000,z100,Tooldata_TCP_ATI\WObj:=Workobject_ruby;
	    MoveL Target_360,v1000,z100,Tooldata_TCP_ATI\WObj:=Workobject_ruby;
	    MoveL Target_370,v1000,z100,Tooldata_TCP_ATI\WObj:=Workobject_ruby;
	    MoveL Target_380,v1000,z100,Tooldata_TCP_ATI\WObj:=Workobject_ruby;
	    MoveL Target_390,v1000,z100,Tooldata_TCP_ATI\WObj:=Workobject_ruby;
	    MoveL Target_400,v1000,z100,Tooldata_TCP_ATI\WObj:=Workobject_ruby;
	    MoveL Target_410,v1000,z100,Tooldata_TCP_ATI\WObj:=Workobject_ruby;
	    MoveL Target_420,v1000,z100,Tooldata_TCP_ATI\WObj:=Workobject_ruby;
	    MoveL Target_430,v1000,z100,Tooldata_TCP_ATI\WObj:=Workobject_ruby;
	    MoveJ Target_440,v1000,z100,Tooldata_TCP_ATI\WObj:=Workobject_ruby;
	    MoveJ Target_450,v1000,z100,Tooldata_TCP_ATI\WObj:=Workobject_ruby;
	    MoveL Target_460,v1000,z100,Tooldata_TCP_ATI\WObj:=Workobject_ruby;
	    MoveL Target_470,v1000,z100,Tooldata_TCP_ATI\WObj:=Workobject_ruby;
	    MoveL Target_480,v1000,z100,Tooldata_TCP_ATI\WObj:=Workobject_ruby;
	    MoveL Target_490,v1000,z100,Tooldata_TCP_ATI\WObj:=Workobject_ruby;
	    MoveL Target_500,v1000,z100,Tooldata_TCP_ATI\WObj:=Workobject_ruby;
	    MoveJ Target_500_2,v1000,z100,Tooldata_TCP_ATI\WObj:=Workobject_ruby;
	    MoveJ Target_500_2_2,v1000,z100,Tooldata_TCP_ATI\WObj:=Workobject_ruby;
	    MoveJ Target_510,v1000,z100,Tooldata_TCP_ATI\WObj:=Workobject_ruby;
	    MoveJ Target_520,v1000,z100,Tooldata_TCP_ATI\WObj:=Workobject_ruby;
	    MoveC Target_530,Target_540,v1000,z100,Tooldata_TCP_ATI\WObj:=Workobject_ruby;
	    MoveC Target_550,Target_560,v1000,z100,Tooldata_TCP_ATI\WObj:=Workobject_ruby;
	    MoveJ Target_570,v1000,z100,Tooldata_TCP_ATI\WObj:=Workobject_ruby;
	    MoveJ Target_580_3,v1000,z100,Tooldata_TCP_ATI\WObj:=Workobject_ruby;
	    MoveJ Target_740,v1000,z100,Tooldata_TCP_ATI\WObj:=Workobject_ruby;
	    MoveJ Target_580_3_2,v1000,z100,Tooldata_TCP_ATI\WObj:=Workobject_ruby;
	    MoveJ Target_580,v1000,z100,Tooldata_TCP_ATI\WObj:=Workobject_ruby;
	    MoveJ Target_590,v1000,z100,Tooldata_TCP_ATI\WObj:=Workobject_ruby;
	    MoveL Target_600,v1000,z100,Tooldata_TCP_ATI\WObj:=Workobject_ruby;
	    MoveL Target_610,v1000,z100,Tooldata_TCP_ATI\WObj:=Workobject_ruby;
	    MoveL Target_620,v1000,z100,Tooldata_TCP_ATI\WObj:=Workobject_ruby;
	    MoveL Target_630,v1000,z100,Tooldata_TCP_ATI\WObj:=Workobject_ruby;
	    MoveL Target_640,v1000,z100,Tooldata_TCP_ATI\WObj:=Workobject_ruby;
	    MoveL Target_650,v1000,z100,Tooldata_TCP_ATI\WObj:=Workobject_ruby;
	    MoveL Target_660,v1000,z100,Tooldata_TCP_ATI\WObj:=Workobject_ruby;
	    MoveL Target_670,v1000,z100,Tooldata_TCP_ATI\WObj:=Workobject_ruby;
	    MoveL Target_680,v1000,z100,Tooldata_TCP_ATI\WObj:=Workobject_ruby;
	    MoveL Target_690,v1000,z100,Tooldata_TCP_ATI\WObj:=Workobject_ruby;
	    MoveL Target_700,v1000,z100,Tooldata_TCP_ATI\WObj:=Workobject_ruby;
	    MoveL Target_710,v1000,z100,Tooldata_TCP_ATI\WObj:=Workobject_ruby;
	    MoveL Target_720,v1000,z100,Tooldata_TCP_ATI\WObj:=Workobject_ruby;
	    MoveL Target_730,v1000,z100,Tooldata_TCP_ATI\WObj:=Workobject_ruby;
	    MoveJ Target_730_2,v1000,z100,Tooldata_TCP_ATI\WObj:=Workobject_ruby;
	    MoveJ Target_130_2,v500,z100,Flansa_Cuplare\WObj:=Workobject_ruby;
	    MoveJ Target_120_2,v500,z100,Flansa_Cuplare\WObj:=Workobject_ruby;
	    MoveJ Target_110_2,v500,z100,Flansa_Cuplare\WObj:=Workobject_ruby;
	    MoveJ Target_100,v500,z100,Flansa_Cuplare\WObj:=Workobject_ruby;
	ENDPROC
	PROC Path_20()

	ENDPROC
	PROC Path_Skye()
	    MoveJ Target_90_2_2_3_2_2_2_2,v500,z100,Flansa_Cuplare\WObj:=Workobject_Skye;
	    MoveJ Target_100_2,v500,z100,Flansa_Cuplare\WObj:=Workobject_Skye;
	    MoveJ Target_110_3,v500,z100,Flansa_Cuplare\WObj:=Workobject_Skye;
	    MoveJ Target_120_3,v500,z100,Flansa_Cuplare\WObj:=Workobject_Skye;
	    MoveJ Target_130_3,v500,z50,Flansa_Cuplare\WObj:=Workobject_Skye;
	    MoveJ Target_260_2,v100,z50,Flansa_Cuplare\WObj:=Workobject_Skye;
	    MoveL Target_270_2,v200,z50,Flansa_Cuplare\WObj:=Workobject_Skye;
	    MoveL Target_320_2,v1000,z100,Flansa_Cuplare\WObj:=Workobject_Skye;
	    MoveL Target_350_2,v300,z30,Flansa_Cuplare\WObj:=Workobject_Skye;
	    MoveJ Target_360_2,v300,z30,Flansa_Cuplare\WObj:=Workobject_Skye;
	    MoveJ Target_370_2,v300,z30,Flansa_Cuplare\WObj:=Workobject_Skye;
	    MoveL Target_400_2,v300,z30,Flansa_Cuplare\WObj:=Workobject_Skye;
	    MoveJ Target_450_2,v300,z30,Flansa_Cuplare\WObj:=Workobject_Skye;
	    MoveL Target_460_2,v300,z30,Flansa_Cuplare\WObj:=Workobject_Skye;
	    MoveL Target_490_2,v300,z30,Flansa_Cuplare\WObj:=Workobject_Skye;
	    MoveL Target_500_3,v300,z30,Flansa_Cuplare\WObj:=Workobject_Skye;
	    MoveJ Target_740_2,v400,z20,Flansa_Cuplare\WObj:=Workobject_Skye;
	    MoveJ Target_590_2,v300,z30,Flansa_Cuplare\WObj:=Workobject_Skye;
	    MoveL Target_600_2,v300,z30,Flansa_Cuplare\WObj:=Workobject_Skye;
	    MoveJ Target_630_2,v300,z30,Flansa_Cuplare\WObj:=Workobject_Skye;
	    MoveJ Target_660_2,v300,z30,Flansa_Cuplare\WObj:=Workobject_Skye;
	    MoveL Target_670_2,v300,z30,Flansa_Cuplare\WObj:=Workobject_Skye;
	    MoveJ Target_700_2,v300,z30,Flansa_Cuplare\WObj:=Workobject_Skye;
	    MoveJ Target_710_2,v300,z30,Flansa_Cuplare\WObj:=Workobject_Skye;
	    MoveL Target_730_3,v300,z30,Flansa_Cuplare\WObj:=Workobject_Skye;
	    MoveJ Target_730_2_2,v300,z30,Flansa_Cuplare\WObj:=Workobject_Skye;
	    MoveJ Target_130_2_2,v300,z30,Flansa_Cuplare\WObj:=Workobject_Skye;
	ENDPROC
	PROC Path_karma()
	    MoveJ Target_130_2_2_2,v400,z30,Flansa_Cuplare\WObj:=Workobject_karma;
	    MoveJ Target_90_2_2_2,v400,z30,Flansa_Cuplare\WObj:=Workobject_karma;
	    MoveJ Target_90_2_3,v400,z30,Tooldata_TCP_VAC\WObj:=Workobject_karma;
	    MoveJ Target_90_2_4,v400,z30,Tooldata_TCP_VAC\WObj:=Workobject_karma;
	    MoveJ Target_90_3,v400,z30,Tooldata_TCP_VAC\WObj:=Workobject_karma;
	    MoveJ Target_80_3,v400,z30,Tooldata_TCP_VAC\WObj:=Workobject_karma;
	    MoveJ Target_80_2_2,v400,z30,Tooldata_TCP_VAC\WObj:=Workobject_karma;
	    MoveJ Target_70_2,v400,z30,Tooldata_TCP_VAC\WObj:=Workobject_karma;
	    MoveJ Target_30_2,v150,z10,Tooldata_TCP_VAC\WObj:=Workobject_karma;
	    MoveL Target_30_3_2,v150,z10,Tooldata_TCP_VAC\WObj:=Workobject_karma;
	    MoveL Target_30_2_2,v150,z10,Tooldata_TCP_VAC\WObj:=Workobject_karma;
	    MoveJ Target_30_2_3,v300,z30,Tooldata_TCP_VAC\WObj:=Workobject_karma;
	    MoveJ Target_30_2_3_2,v300,z30,Tooldata_TCP_VAC\WObj:=Workobject_karma;
	    MoveJ Target_30_2_3_2_2,v300,z30,Tooldata_TCP_VAC\WObj:=Workobject_karma;
	    MoveJ Target_30_2_3_2_2_2,v300,z30,Tooldata_TCP_VAC\WObj:=Workobject_karma;
	    MoveJ Target_30_2_3_2_2_2_2,v300,z30,Tooldata_TCP_VAC\WObj:=Workobject_karma;
	    MoveJ Target_30_2_3_2_2_2_2_2,v300,z30,Tooldata_TCP_VAC\WObj:=Workobject_karma;
	    MoveJ Target_30_2_3_2_2_2_2_2_2,v300,z30,Tooldata_TCP_VAC\WObj:=Workobject_karma;
	ENDPROC
ENDMODULE
